{attribute 'qualified_only'}
{attribute 'strict'}
{attribute 'to_string'}
TYPE E_LIST_CHECK :
(
	NULL,
  REFERENCE_CTRL_INVALID := 9000,
  REFERENCE_STATE_INVALID,
  REFERENCE_DATA_INPUT_INVALID,
  REFERENCE_DATA_OUTPUT_INVALID,

  CHECK_DONE              := 10000
);
END_TYPE

(* stored: Version 1.1.0.1, ProductVersion 3.1.4026.18
   DUT E_LIST_CHECK: Id {cab5ef07-4263-4d6e-ba24-77d34271d55b} *)
